# EPICS StreamDevice protocol: protocol/ELSE-SATURN5702.proto
# ELSE-SATURN5702.proto

# Communication protocol for ELSE Nuclear probes (ICP-T-PF and LUPIN 5401 BF3-NP models) and SATURN

# Protocol terminator character

Terminator = LF;

# Gamma

getGamma {
    out "RAD_E_Gamma?";
    in "%f";
}

# Neutron

getNeutron {
    out "RAD_E_Neutron?";
    in "%f";
}

# Total dose rate

getTotalDoseRate {
    out "RAD_E_Total?";
    in "%f";
}

# Total Integral

getIntegral {
    out "RAD_E_Integral?";
    in "%f";
}

# Total Integral Gamma

getIntegralGamma {
    out "RAD_E_IntegralGamma?";
    in "%f";
}

# Total Integral Neutron

getIntegralNeutron {
    out "RAD_E_IntegralNeutron?";
    in "%f";
}
